// TIA Portal V20 export
TYPE "LKinCtrl_typeMovePathTracking"
// stored: Access Published
   STRUCT
      selectedPath { ExternalAccessible := 'False'; ExternalVisible := 'False'; ExternalWritable := 'False'} : DInt;
      status { ExternalAccessible := 'False'; ExternalVisible := 'False'; ExternalWritable := 'False'} : Word;
      activeCmdNo { ExternalAccessible := 'False'; ExternalVisible := 'False'; ExternalWritable := 'False'} : DInt;
      remainingDistanceActCmd { ExternalAccessible := 'False'; ExternalVisible := 'False'; ExternalWritable := 'False'} : LReal;
   END_STRUCT;
END_TYPE
